VAR_GLOBAL
	instEmitterConveyorFeedIn	:	FactoryIO.FB_Emitter;	//Instanz FB_Emitter Zufuehrband Einlauf
	
END_VAR

(* stored: Version 1.1.0.1
   GVL Emitter: Id {546306e6-6e6a-46b1-83d9-446781607f98} *)
